TYPE DUT_GetResourcesByName :
STRUCT
	return_value	: DINT;
	ResourceName	: STRING(50);
END_STRUCT
END_TYPE

(* stored: Version 1.1.0.1, ProductVersion 3.1.4024.15
   DUT DUT_GetResourcesByName: Id {7501f314-633a-4f9e-a968-b59ff5c841f0} *)
